{attribute 'no_explicit_call' := 'do not call this POU directly'}
FUNCTION_BLOCK FINAL FB_LoggedEventsSortAscending IMPLEMENTS I_LoggedEventsSort
VAR_INPUT
END_VAR
VAR_OUTPUT
END_VAR
VAR
END_VAR

METHOD Sort : HRESULT
VAR_IN_OUT
	aLoggedEvents	: T_LoggedEvents;
END_VAR
{warning 'TODO: Implement sorting in ascending order'}
Sort := S_OK;
END_METHOD

END_FUNCTION_BLOCK

(* stored: Version 1.1.0.1, ProductVersion 3.1.4024.12
   POU FB_LoggedEventsSortAscending: Id {e5abad23-e6bf-4bcc-b380-454d6be765af}, SpecialFunc None
   Method Sort: Id {391850cf-d80f-4dd7-a0d1-6bff01aa081d} *)
